// TIA Portal V16 export
// export: Created 2023-03-29T11:04:34.9975053Z, ExportSetting WithDefaults, DisplayName Totally Integrated Automation Portal, DisplayVersion V16 Update 6, DisplayName TIA Portal Version Control Interface, DisplayVersion V16 Update 2, DisplayName TIA Portal Openness, DisplayVersion V16 Update 6, DisplayName STEP 7 Professional, DisplayVersion V16 Update 6, DisplayName STEP 7 Safety, DisplayVersion V16, DisplayName WinCC Advanced, DisplayVersion V16 Update 6
DATA_BLOCK "EX012_IDB8_ErrorHandling"   // DB104
VERSION : 0.1
// stored: AutoNumber false, DBAccessibleFromOPCUA true, InstanceOfName EX012_ErrorHandling, InstanceOfType FB
"EX012_ErrorHandling"
   // VAR_INPUT
   //    LED : Int;
   //    CounterError : USInt;
   // END_VAR
   // VAR_OUTPUT
   //    RedLED : Bool;
   // END_VAR
   // VAR
   //    tempCounterDiagStatus : USInt;
   //    tempCounterError : USInt;
   // END_VAR
BEGIN
END_DATA_BLOCK
